{attribute 'OPC.UA.DA.StructuredType' := '1'}
FUNCTION_BLOCK FB_Sensor_GrowMedium_EC EXTENDS FB_BaseSensor IMPLEMENTS I_Device, I_Sensor

VAR
	
	bCAL: BOOL := FALSE;
	
	eSMState: (WAIT, CAL_LOW, CAL_HIGH, CALC_CORRECTION) := WAIT;

END_VAR
	
VAR PERSISTENT ;
	nECLOW_val: REAL;
	nECHIGH_val: REAL;
	
	nCurveGradient: REAL := 0.625; // 
	nCurveOffset: REAL := -2.5; // Defaults
END_VAR

calculate();
filter();

// Detect if any buttons in ignition have been pressed for Calibration
IF bCAL THEN 
	bCAL := FALSE;
	CASE eSMState OF
		WAIT:
			eSMState := CAL_LOW;
		CAL_LOW:
			eSMState := CAL_HIGH;
		CAL_HIGH:
			eSMState := CALC_CORRECTION;
	END_CASE
END_IF


CASE eSMState OF 
	WAIT:
		// wait here for a calibration command to be received
		eState := E_DeviceState.RUNNING;


	CAL_LOW:
		nECLOW_val := nMeasuredCurrent;
		eState := E_DeviceState.CAL_STEP1;

	CAL_HIGH:
		nECHIGH_val := nMeasuredCurrent;
		eState := E_DeviceState.CAL_STEP2;
	
	CALC_CORRECTION:
		nCurveGradient := ((1413.0-84.0)/1000.0) / (nECHIGH_val - nECLOW_val);
		nCurveOffset := (84.0/1000.0) - (nCurveGradient * nECLOW_val);
		eSMState := WAIT;
		eState := E_DeviceState.CAL_STEP3;
		
		
END_CASE

METHOD PRIVATE calculate : BOOL
VAR_INPUT
	
END_VAR
nMeasuredCurrent := (INT_TO_REAL(nRawInput)/GVL.nMaxADCOutput)*16.0 + 4.0; // in mA

// nCurrentValue := (nCurveGradient * nMeasuredCurrent) + nCurveOffset;

nCurrentValue := (nCurveGradient * nFilteredCurrent) + nCurveOffset; // delete this eventually
END_METHOD

METHOD calibrate : BOOL
VAR_INPUT
	
END_VAR
bCAL := TRUE;
END_METHOD

{warning 'add method implementation '}
METHOD disable : BOOL
bEnable := FALSE;
END_METHOD

{warning 'add method implementation '}
METHOD enable : BOOL
bEnable := TRUE;
END_METHOD

{warning 'add method implementation '}
METHOD FB_init : BOOL
VAR_INPUT
	(* if TRUE, the retain variables are initialized (warm start / cold start)*)
	bInitRetains	: BOOL;
	(* if TRUE, the instance afterwards gets moved into the copy code (online change)*)
	bInCopyCode	: BOOL;
	
	SensorID	: STRING(80);
	SensorDescr	: STRING(255);
	SensorType	: E_SensorType;
END_VAR
sID := SensorID;
sDescr := SensorDescr;
eSensorType := SensorType;
END_METHOD

{warning 'add method implementation '}
METHOD getType : E_SensorType
getType := eSensorType;
END_METHOD

{warning 'add method implementation '}
METHOD getValue : REAL
getValue := nCurrentValue;
END_METHOD

{warning 'add method implementation '}
METHOD write : BOOL
// use this method to initiated a hardware read from assigned IO if required
END_METHOD

END_FUNCTION_BLOCK

(* stored: Version 1.1.0.1, ProductVersion 3.1.4024.12
   POU FB_Sensor_GrowMedium_EC: Id {6d977c64-a1ae-4886-9cdc-a9064bbc6a2b}, SpecialFunc None
   Method calculate: Id {831cb252-8f34-4832-9284-fd14917d1241}
   Method calibrate: Id {da174f71-6a65-4e3f-a82a-f9c01cd8c680}
   Method disable: Id {e19b1335-0c0d-44b7-82c4-9f39250b3a0f}
   Method enable: Id {9d885b96-fa1d-4ee5-88b6-e2fa10e951d1}
   Method FB_init: Id {ce2b81a2-af48-4dcd-887a-bd3d45f44de9}
   Method getType: Id {7c514f1e-01ea-42e9-8a22-dbeea87bb549}
   Method getValue: Id {eae2c1bb-0fb4-4e04-bffd-69a30bc80951}
   Method write: Id {117a4a12-0f5f-4db0-b368-397afe6bbd7f} *)
